{attribute 'qualified_only'}
{attribute 'strict'}

//-----------------------------------------------------------------------------------------
//
//                  				ENUM_Fan_Type
//
//						Enumération des types de ventilateur(s)			
//-----------------------------------------------------------------------------------------
//
//Auteur: G.GOETZ
//Création: 20.01.2026
//Dernière modification : 20.01.2026 (G.GOETZ)
//       			
//-----------------------------------------------------------------------------------------
//
//     							Liste des modifications  	
//
// 20.01.2026 (G.GOETZ) -> Création		
//-----------------------------------------------------------------------------------------

TYPE ENUM_Fan_Type :
(
	(*Unknow := 0 , // Unknow type*)
	PWM := 1 // With PWM type
);
END_TYPE

(* stored: Version 1.1.0.1, ProductVersion 3.1.4024.13
   DUT ENUM_Fan_Type: Id {37285349-f9d7-4688-ac1d-68defd7adea2} *)
